Universal Robots PolyScope program: c_full_bow.urp

Program c_full_bow (installation=string_planes directory=/programs/strings createdIn=5.17.3 lastSavedIn=5.17.3 robotSerialNumber=20245501435)
Calibrated DH parameters: a=[0.000154, -0.137004, -0.385524, -0.00002, 0.000092, 0]; d=[0.162441, 211.794786, -230.585024, 18.923638, 0.099786, 0.09951]; alpha=[1.569493, -0.001902, 0.003874, 1.570111, -1.570167, 0]; deltaTheta=[0, -1.242934, 1.056292, 0.186646, 0.000002, 0.000001]
InitVariablesNode
Robot Program (runOnlyOnce=false)
  MoveL speed 250 mm/s, acceleration 1200 mm/s^2 (useActiveTCP=true) feature=Base
    Waypoint Waypoint_4: TCP in base x=343.41 y=632.837 z=65.917 mm, rx=-1.6485 ry=-1.4729 rz=0.5687 rad; joints [-133.534, -25.075, 76.855, -110.444, -40.013, -141.74] deg; TCP offset x=28.21 y=-96.107 z=-99.69 mm, rx=0 ry=0 rz=0 rad
    Waypoint Waypoint_6: TCP in base x=239.865 y=239.465 z=-96.417 mm, rx=-1.496 ry=-1.6066 rz=0.56 rad; joints [-162.973, -14.775, 123.07, -145.576, -63.187, -180.115] deg
  MoveL speed 250 mm/s, acceleration 1200 mm/s^2 (useActiveTCP=true) feature=Base
    Waypoint Waypoint_6: TCP in base x=239.865 y=239.465 z=-96.417 mm, rx=-1.496 ry=-1.6066 rz=0.56 rad; joints [-162.973, -14.775, 123.07, -145.576, -63.187, -180.115] deg
    Waypoint Waypoint_4: TCP in base x=343.41 y=632.837 z=65.917 mm, rx=-1.6485 ry=-1.4729 rz=0.5687 rad; joints [-133.534, -25.075, 76.855, -110.444, -40.013, -141.74] deg
  Wait Sleep waitTime=300
  bow_dir := True
  note_dur := 1
  Timer (action=Start) variable(name=timer_1)
  If bow_dir≟ True
    MoveL speed 250 mm/s, acceleration 1200 mm/s^2 (useActiveTCP=true) feature=Base
      Waypoint Waypoint_6: TCP in base x=239.865 y=239.465 z=-96.417 mm, rx=-1.496 ry=-1.6066 rz=0.56 rad; joints [-162.973, -14.775, 123.07, -145.576, -63.187, -180.115] deg
        Until EXPRESSION (allowActions=false) ExpressionBranch=timer_1≟note_dur
  Else 
    MoveL speed 250 mm/s, acceleration 1200 mm/s^2 (useActiveTCP=true) feature=Base
      Waypoint Waypoint_4: TCP in base x=343.41 y=632.837 z=65.917 mm, rx=-1.6485 ry=-1.4729 rz=0.5687 rad; joints [-133.534, -25.075, 76.855, -110.444, -40.013, -141.74] deg
        Until EXPRESSION (allowActions=false) ExpressionBranch=timer_1≟note_dur
  SuppressedNode
    MoveL speed 250 mm/s, acceleration 1200 mm/s^2 (useActiveTCP=true) feature=Base
      Waypoint Waypoint_4: TCP in base x=245.284 y=570.71 z=53.266 mm, rx=-1.8425 ry=-1.3918 rz=0.0687 rad; joints [-132.226, -24.798, 96.314, -169.322, -42.692, -112.607] deg
      Waypoint Waypoint_1: TCP in base x=195.249 y=411.456 z=21.268 mm, rx=-1.7342 ry=-1.5169 rz=0.4322 rad; joints [-140.231, -30.936, 122.536, -154.99, -45.802, -143.197] deg
      Waypoint Waypoint_6: TCP in base x=152.636 y=275.824 z=-5.984 mm, rx=-1.6122 ry=-1.6008 rz=0.7404 rad; joints [-153.501, -26.653, 138.52, -151.348, -62.645, -165.795] deg
  Timer (action=Stop) variable=timer_1
  Timer (action=Reset) variable=timer_1
